TYPE DUT_Robot2 :
STRUCT
		xMaterialOnOff : BOOL ;
        stProduct :ARRAY[1..5] OF DUT_PartStatus ;
END_STRUCT
END_TYPE

(* stored: Version 1.1.0.1, ProductVersion 3.1.4024.9
   DUT DUT_Robot2: Id {e4fca855-80db-48cc-9ba6-4b45ea2879c9} *)
